FUNCTION_BLOCK MotionControl
VAR_INPUT
END_VAR
VAR_OUTPUT
END_VAR
VAR
	cncChannnelHandler	:TC_CNC;
	refAxis		: AXIS_REF;
END_VAR

ACTION AxisControl:

END_ACTION

METHOD GetPosition : DWORD
VAR_INPUT
END_VAR
END_METHOD

METHOD setAxis : BOOL
VAR_INPUT
	refToAxis		:AXIS_REF;
END_VAR
END_METHOD

METHOD SetParams : BOOL
VAR_INPUT
END_VAR
END_METHOD

METHOD SetPosition : BOOL
VAR_INPUT
END_VAR
END_METHOD

END_FUNCTION_BLOCK

(* stored: Version 1.1.0.1, ProductVersion 3.1.4024.11
   POU MotionControl: Id {1e33ec8f-67b8-4708-8ed2-209b19dae61f}, SpecialFunc None
   Action AxisControl: Id {935ac1fc-1b1d-4d8e-8e68-82d4529718fc}
   Method GetPosition: Id {fd1d2b8c-fc3a-484e-bd80-052e41828328}
   Method setAxis: Id {8ed7fae7-762a-4c5c-a6db-e0eed52615e9}
   Method SetParams: Id {a15fad5c-e4f7-4216-8d35-33473220a766}
   Method SetPosition: Id {dc7dbf2f-ab9e-4917-9eba-cd2f69ccd871} *)
